{attribute 'qualified_only'}
VAR_GLOBAL
	MPA01: DUT_DoubleActPneumaticActuator;
	MPA02: DUT_DoubleActPneumaticActuator;
	MPA03: DUT_DoubleActPneumaticActuator;
	MPA04: DUT_DoubleActPneumaticActuator;
END_VAR

(* stored: Version 1.1.0.1, ProductVersion 3.1.4022.18
   GVL RTDSL0: Id {ac721235-6abd-4ba5-afeb-f19d34581d05} *)
